FUNCTION_BLOCK FB_ESSMonitoringMCU6001a EXTENDS FB_ESSMonitoringBase
VAR
    //Outputs
    {attribute 'TcLinkTo' := 'TIID^Device 1 (EtherCAT)^KF201 (EK1200)^KF206 (EL2014)^DIG Outputs^Channel 1^Output'}
    bStatusLED AT %Q*: BOOL;
    {attribute 'TcLinkTo' := 'TIID^Device 1 (EtherCAT)^KF201 (EK1200)^KF205 (EL2014)^DIG Outputs^Channel 4^Output'}
    bAcknowledgeLED AT %Q*: BOOL;
    {attribute 'TcLinkTo' := 'TIID^Device 1 (EtherCAT)^KF201 (EK1200)^KF206 (EL2014)^DIG Outputs^Channel 2^Output'}
    bEStopLED AT %Q*: BOOL;
    {attribute 'TcLinkTo' := 'TIID^Device 1 (EtherCAT)^KF201 (EK1200)^KF206 (EL2014)^DIG Outputs^Channel 4^Output'}
    bErrorLED AT %Q*: BOOL;

    //Inputs
    {attribute 'TcLinkTo' := 'TIID^Device 1 (EtherCAT)^KF201 (EK1200)^KF204 (EL1808)^Channel 1^Input'}
    b24VDC1_OK AT %I*: BOOL;
    {attribute 'TcLinkTo' := 'TIID^Device 1 (EtherCAT)^KF201 (EK1200)^KF204 (EL1808)^Channel 2^Input'}
    b24VDC2_OK AT %I*: BOOL;
    {attribute 'TcLinkTo' := 'TIID^Device 1 (EtherCAT)^KF201 (EK1200)^KF204 (EL1808)^Channel 3^Input'}
    b24VDC3_OK AT %I*: BOOL;
    {attribute 'TcLinkTo' := 'TIID^Device 1 (EtherCAT)^KF201 (EK1200)^KF204 (EL1808)^Channel 4^Input'}
    b48VDC1_OK AT %I*: BOOL;
    {attribute 'TcLinkTo' := 'TIID^Device 1 (EtherCAT)^KF201 (EK1200)^KF203 (EL1808)^Channel 1^Input'}
    bFuse1_OK AT %I*: BOOL;
    {attribute 'TcLinkTo' := 'TIID^Device 1 (EtherCAT)^KF201 (EK1200)^KF203 (EL1808)^Channel 2^Input'}
    bFuse2_OK AT %I*: BOOL;
    {attribute 'TcLinkTo' := 'TIID^Device 1 (EtherCAT)^KF201 (EK1200)^KF203 (EL1808)^Channel 3^Input'}
    bFuse3_OK AT %I*: BOOL;
    {attribute 'TcLinkTo' := 'TIID^Device 1 (EtherCAT)^KF201 (EK1200)^KF203 (EL1808)^Channel 7^Input'}
    bSPD_OK AT %I*: BOOL;
    {attribute 'TcLinkTo' := 'TIID^Device 1 (EtherCAT)^KF201 (EK1200)^KF203 (EL1808)^Channel 8^Input'}
    bDoorClosed AT %I*: BOOL;
    {attribute 'TcLinkTo' := 'TIID^Device 1 (EtherCAT)^KF201 (EK1200)^KF204 (EL1808)^Channel 5^Input'}
    bEStop1Released AT %I*: BOOL;
    {attribute 'TcLinkTo' := 'TIID^Device 1 (EtherCAT)^KF201 (EK1200)^KF204 (EL1808)^Channel 6^Input'}
    bSTO1Released AT %I*: BOOL;
    {attribute 'TcLinkTo' := 'TIID^Device 1 (EtherCAT)^KF201 (EK1200)^KF204 (EL1808)^Channel 8^Input'}
    bAcknowledgeButton AT %I*: BOOL;
    {attribute 'TcLinkTo' := 'TIID^Device 1 (EtherCAT)^KF201 (EK1200)^KF207 (EL3214)^RTD Inputs Channel 1^Value'}
    nTemp1 AT %I*: INT;
    {attribute 'TcLinkTo' := 'TIID^Device 1 (EtherCAT)^KF201 (EK1200)^KF207 (EL3214)^RTD Inputs Channel 2^Value'}
    nTemp2 AT %I*: INT;
    {attribute 'TcLinkTo' := 'TIID^Device 1 (EtherCAT)^KF201 (EK1200)^KF207 (EL3214)^RTD Inputs Channel 3^Value'}
    nTemp3 AT %I*: INT;
    {attribute 'TcLinkTo' := 'TIID^Device 1 (EtherCAT)^KF201 (EK1200)^KF207 (EL3214)^RTD Inputs Channel 4^Value'}
    nTemp4 AT %I*: INT;
    {attribute 'TcLinkTo' := 'TIID^Device 1 (EtherCAT)^Inputs^DevState'}
    nEcMasterDevState AT %I*: UINT;

    //Shutter OP
    {attribute 'TcLinkTo' := 'TIID^Device 1 (EtherCAT)^KF201 (EK1200)^KF217 (EK1521)^KF01 (EK1501-0100)^KF02 (EL1808)^Channel 1^Input'}
    bShutterOPFuse1_OK AT %I*: BOOL;
    {attribute 'TcLinkTo' := 'TIID^Device 1 (EtherCAT)^KF201 (EK1200)^KF217 (EK1521)^KF01 (EK1501-0100)^KF02 (EL1808)^Channel 2^Input'}
    bShutterOPFuse2_OK AT %I*: BOOL;
    {attribute 'TcLinkTo' := 'TIID^Device 1 (EtherCAT)^KF201 (EK1200)^KF217 (EK1521)^KF01 (EK1501-0100)^KF02 (EL1808)^Channel 3^Input'}
    bShutterOP24VDC1_OK AT %I*: BOOL;
    {attribute 'TcLinkTo' := 'TIID^Device 1 (EtherCAT)^KF201 (EK1200)^KF217 (EK1521)^KF01 (EK1501-0100)^KF02 (EL1808)^Channel 4^Input'}
    bShutterOPSPD_OK AT %I*: BOOL;
END_VAR

SUPER^();

METHOD mLink
// Input variables
AcknowledgeButton := bAcknowledgeButton;
EStopReleased := bEStop1Released;
EcMasterDevState := nEcMasterDevState;

// Output variables
bAcknowledgeLED := AcknowledgeLED;
bStatusLED := StatusLED;
bEStopLED := EStopLED;
bErrorLED := ErrorLED;
END_METHOD

METHOD mSetResetAlarmsLeds
VAR_INST
    index: UINT;
    aDeadBandActive: ARRAY [1..4] OF BOOL;
    nDeadBandTemperature: INT := 3;
    aTemperatureAlarm: ARRAY [1..4] OF BOOL;
END_VAR
mSetReset(stAlarmList := aAlarmList[1], bOk := b24VDC1_OK);
mSetReset(stAlarmList := aAlarmList[2], bOk := b24VDC2_OK);
mSetReset(stAlarmList := aAlarmList[3], bOk := b24VDC3_OK);

mSetReset(stAlarmList := aAlarmList[4], bOk := b48VDC1_OK);

mSetReset(stAlarmList := aAlarmList[9], bOk := bSPD_OK);
mSetReset(stAlarmList := aAlarmList[10], bOk := bDoorClosed);

mSetReset(stAlarmList := aAlarmList[11], bOk := bFuse1_OK);
mSetReset(stAlarmList := aAlarmList[12], bOk := bFuse2_OK);
mSetReset(stAlarmList := aAlarmList[13], bOk := bFuse3_OK);

mSetReset(stAlarmList := aAlarmList[19], bOk := bEStop1Released);
//mSetReset(stAlarmList := aAlarmList[20], bOk := bSTO1Released);

mSetReset(stAlarmList := aAlarmList[27], bOk := NOT bEcMasterError);
mSetReset(stAlarmList := aAlarmList[28], bOk := NOT bSlaveStateNotOP);
mSetReset(stAlarmList := aAlarmList[29], bOk := NOT bSlaveLinkError);
mSetReset(stAlarmList := aAlarmList[30], bOk := NOT bCycleTimeExceeded);
mSetReset(stAlarmList := aAlarmList[31], bOk := NOT bCPUOverloaded);

mSetReset(stAlarmList := aAlarmList[34], bOk := bShutterOPFuse1_OK);
mSetReset(stAlarmList := aAlarmList[35], bOk := bShutterOPFuse2_OK);
mSetReset(stAlarmList := aAlarmList[36], bOk := bShutterOP24VDC1_OK);
mSetReset(stAlarmList := aAlarmList[37], bOk := bShutterOPSPD_OK);


aTemperatureAlarm[1] :=
    nTemp1 > nMAX_TEMP
    OR (aDeadBandActive[1] AND nTemp1 > (nMAX_TEMP - nDeadBandTemperature));
aDeadBandActive[1] := aTemperatureAlarm[1];
mSetReset(stAlarmList := aAlarmList[23], bOk := NOT aTemperatureAlarm[1]);

aTemperatureAlarm[2] :=
    nTemp2 > nMAX_TEMP
    OR (aDeadBandActive[2] AND nTemp2 > (nMAX_TEMP - nDeadBandTemperature));
aDeadBandActive[2] := aTemperatureAlarm[2];
mSetReset(stAlarmList := aAlarmList[24], bOk := NOT aTemperatureAlarm[2]);

aTemperatureAlarm[3] :=
    nTemp3 > nMAX_TEMP
    OR (aDeadBandActive[3] AND nTemp3 > (nMAX_TEMP - nDeadBandTemperature));
aDeadBandActive[3] := aTemperatureAlarm[3];
mSetReset(stAlarmList := aAlarmList[25], bOk := NOT aTemperatureAlarm[3]);

aTemperatureAlarm[4] :=
    nTemp4 > nMAX_TEMP
    OR (aDeadBandActive[4] AND nTemp4 > (nMAX_TEMP - nDeadBandTemperature));
aDeadBandActive[4] := aTemperatureAlarm[4];
mSetReset(stAlarmList := aAlarmList[26], bOk := NOT aTemperatureAlarm[4]);
END_METHOD

END_FUNCTION_BLOCK

(* stored: Version 1.1.0.1
   POU FB_ESSMonitoringMCU6001a: Id {61812d1b-8eb2-03ad-1b15-beb88a4506c3}, SpecialFunc None
   Method mLink: Id {98cdd0c2-7af6-02ba-3a8d-c667c75f0bdb}
   Method mSetResetAlarmsLeds: Id {297e9ae8-2e7e-0581-2e8a-fc9b407c0960} *)
